Staubli VAL3: VelocityCfgMsg.pjx

--- VelocityCfgMsg.pjx ---
Parameters version=s7.8.1 stackSize=5000 millimeterUnit=true
Program file=start.pgx
Program file=stop.pgx
Data file=VelocityCfgMsg.dtx
Type name=Prefix path=Disk://ros_libs/Prefix/Prefix.pjx
Type name=Header path=Disk://ros_libs/Header/Header.pjx
Type name=Body path=Disk://ros_libs/Body/Body.pjx
Type name=VelocityCfg path=../VelocityCfg/VelocityCfg.pjx

--- VelocityCfgMsg.dtx ---
public Prefix prefix
  [0]
    num nLength
    num nData[4]
public Header header
  [0]
    num nMsgType
    num nCommType
    num nReplyCode
    num nData[12]
public Body body
  [0]
    num nData[68]
public VelocityCfg velCfg
  [0]
    num nCmdType
    num nRefFrameVec[6]
    num nToolVec[6]
    num nAccel
    num nVel
    num nTransVel
    num nRotVel

--- start.pgx ---
program start()
begin
  // Copyright (c) 2021, Institute for Factory Automation and Production Systems (FAPS)
  //
  // Licensed under the Apache License, Version 2.0 (the "License");
  // you may not use this file except in compliance with the License.
  // You may obtain a copy of the License at
  //
  //     http://www.apache.org/licenses/LICENSE-2.0
  //
  // Unless required by applicable law or agreed to in writing, software
  // distributed under the License is distributed on an "AS IS" BASIS,
  // WITHOUT WARRANTIES OR CONDITIONS OF ANY KIND, either express or implied.
  // See the License for the specific language governing permissions and
  // limitations under the License.


end
